FUNCTION ck_state_v : INT
VAR_INPUT
	
	data_vision : Vision_int_state;
    
END_VAR
VAR
	ck0 : INT;
	ck1 : INT;
	ck2 : INT;
END_VAR


ck0 := data_vision.Val1;
ck1 := data_vision.Val2;
ck2 := data_vision.Val3;


//IF (ck0=state AND ck1=state AND ck2=state) OR (ck1=state AND ck2=state) OR (ck0=state AND ck2=state) OR (ck0=state AND ck1=state ) THEN
IF ck0 = ck1 THEN
ck_state_v := ck0;	
ELSIF  ck1 = ck2 THEN 
ck_state_v := ck1;	
ELSIF  ck2 = ck0 THEN
ck_state_v := ck2;	
ELSE 
ck_state_v := -1;	
END_IF

END_FUNCTION

(* stored: Version 1.1.0.1, ProductVersion 3.1.4024.4
   POU ck_state_v: Id {04149043-8498-460e-b3b3-29c278d99752}, SpecialFunc None *)
